// TIA Portal project "Plantilla_Prensa" (V17)

(* hardware
DEVICE "S7-1200 station_1"  S7-1200 Station
   slot 0: "Rack_0"  S7-1200 Rack  Rack  V1.0
   slot 1: "PLC_1"  CPU 1214C AC/DC/Rly  6ES7 214-1BG40-0XB0  V4.5
*)

// ===== PLC "PLC_1"  CPU 1214C AC/DC/Rly =====

VAR_GLOBAL   // PLC tag table "Tabla de variables estándar"
   "System_Byte" AT %MB1 : Byte;
   "FirstScan" AT %M1.0 : Bool;
   "DiagStatusUpdate" AT %M1.1 : Bool;
   "AlwaysTRUE" AT %M1.2 : Bool;
   "AlwaysFALSE" AT %M1.3 : Bool;
   "Clock_Byte" AT %MB0 : Byte;
   "Clock_10Hz" AT %M0.0 : Bool;
   "Clock_5Hz" AT %M0.1 : Bool;
   "Clock_2.5Hz" AT %M0.2 : Bool;
   "Clock_2Hz" AT %M0.3 : Bool;
   "Clock_1.25Hz" AT %M0.4 : Bool;
   "Clock_1Hz" AT %M0.5 : Bool;
   "Clock_0.625Hz" AT %M0.6 : Bool;
   "Clock_0.5Hz" AT %M0.7 : Bool;
END_VAR

DATA_BLOCK "Bloque de datos_1"   // DB7
{ S7_Optimized_Access := 'FALSE' }
VERSION : 0.1
   VAR
      Start : Bool;
      Stop : Bool;
      Alarma : Bool;
      Lámpara : Bool;
      Sensor : Bool;
      "Cilindro Retirado" : Bool;
      "Cilindro Extraido" : Bool;
      "Sensor B4" : Bool;
      "Reset General" : Bool;
      "Golpe 2" : Bool;
      Bloqueo : Bool;
      PT : Time;
      ET : Time;
      CV : Int;
      PV : Int;
      ET1 : Time;
      ET2 : Time;
      ET3 : Time;
      "Fin de ciclo" : Bool;
   END_VAR
BEGIN
END_DATA_BLOCK

// folder: System blocks/Program resources

DATA_BLOCK "IEC_Timer_0_DB"   // DB1
{ S7_Optimized_Access := 'TRUE' }
AUTHOR : Simatic
FAMILY : IEC
NAME : IEC_TMR
VERSION : 1.0
// stored: InstanceOfName IEC_TIMER
"IEC_TIMER"
BEGIN
END_DATA_BLOCK

// folder: (top level)

FUNCTION "Bloque_1" : Void   // FC1, LAD
{ S7_Optimized_Access := 'FALSE' }
VERSION : 0.1
BEGIN

REGION Network 1
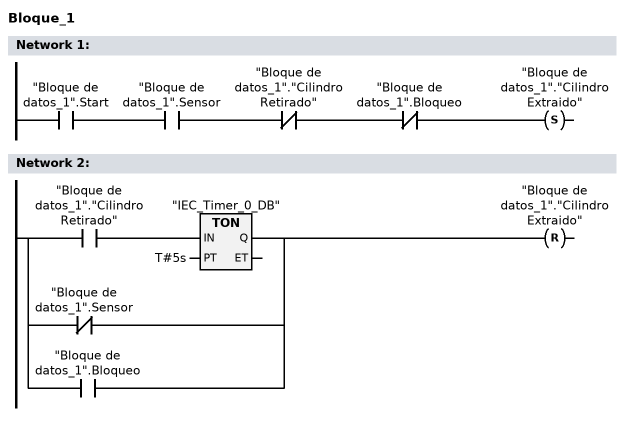
   RUNG wire#powerrail
      Contact( "Bloque de datos_1".Start )
      Contact( "Bloque de datos_1".Sensor )
      I_Contact( "Bloque de datos_1"."Cilindro Retirado" )
      I_Contact( "Bloque de datos_1".Bloqueo )
      S_Coil( "Bloque de datos_1"."Cilindro Extraido" )
   END_RUNG
   // the same network as SCL:
   IF "Bloque de datos_1".Start AND "Bloque de datos_1".Sensor AND NOT "Bloque de datos_1"."Cilindro Retirado" AND NOT "Bloque de datos_1".Bloqueo THEN
       "Bloque de datos_1"."Cilindro Extraido" := TRUE;
   END_IF;
END_REGION

REGION Network 2
   "IEC_Timer_0_DB".TON(IN := "Bloque de datos_1"."Cilindro Retirado", PT := T#5s);
   IF "IEC_Timer_0_DB".Q OR NOT "Bloque de datos_1".Sensor OR "Bloque de datos_1".Bloqueo THEN
       "Bloque de datos_1"."Cilindro Extraido" := FALSE;
   END_IF;
END_REGION
END_FUNCTION

ORGANIZATION_BLOCK "Main"   // OB1, LAD, ProgramCycle
TITLE = "Main Program Sweep (Cycle)"
{ S7_Optimized_Access := 'TRUE' }
VERSION : 0.1
   VAR_INPUT
      Initial_Call : Bool;   // Initial call of this OB
      Remanence : Bool;   // =True, if remanent data are available
   END_VAR
BEGIN

REGION Network 1
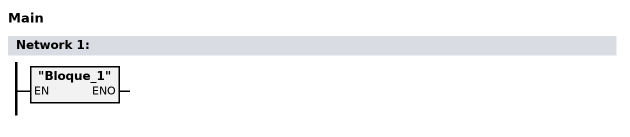
   RUNG wire#powerrail
      "Bloque_1"()
   END_RUNG
   // the same network as SCL:
   "Bloque_1"();
END_REGION
END_ORGANIZATION_BLOCK